// TwinCAT 3 PLC project PrimaryLogic
// ProgramVersion: 3.1.4020.4
// libraries:
//   Tc2_Standard, * (Beckhoff Automation GmbH)
//   Tc2_System, * (Beckhoff Automation GmbH)
//   Tc3_Module, * (Beckhoff Automation GmbH)
// project tree:
//   / PlcTask.TcTTO
//   POUs/ iterator.TcPOU, MAIN.TcPOU

CONFIGURATION PrimaryLogic
    RESOURCE PLC ON TwinCAT3
        TASK PlcTask(INTERVAL := T#50us, PRIORITY := 20);
        PROGRAM MAIN WITH PlcTask : MAIN;
    END_RESOURCE
END_CONFIGURATION

// ---- POUs/MAIN.TcPOU
PROGRAM MAIN
VAR CONSTANT
END_VAR
VAR
	ulimit	:	DINT	:=	1000;
	delay	:	DINT	:=	50;
	assign	:	BOOL	:=	FALSE;
	(**********************)
	arr	:	ARRAY	[0..20000]	OF	iterator;
	cache	:	ARRAY	[0..20000]	OF	DINT;
	noToTest	:	DINT	:= 0;
	count	: DINT	:=0;
	I	:	DINT;
	step	:	BOOL;
END_VAR


IF count < delay-1 THEN
	count := count + 1;
	step :=	FALSE;
ELSE
	count := 0;
	step :=	TRUE;
END_IF

IF step THEN
	IF noToTest < ulimit-1 THEN
		noToTest := noToTest + 1;
	ELSE
		noToTest := 0;
	END_IF
END_IF
// Run noToTest operations
FOR I:=0 TO noToTest BY 1 DO 
	arr[I](increment:=1);
	IF ASSIGN THEN
		cache[I] := arr[i].out;
	END_IF
END_FOR;

END_PROGRAM

// ---- POUs/iterator.TcPOU
FUNCTION_BLOCK iterator
VAR_INPUT
	increment	:	DINT;
END_VAR
VAR_OUTPUT
	out	:	DINT;
END_VAR
VAR
	value	:	DINT	:=0;
	lim	:	DINT :=1000;
END_VAR

IF value < lim THEN
	value := value + increment;
ELSE
	value:= 0;	
END_IF
out := value;

END_FUNCTION_BLOCK
